PROGRAM MAIN
VAR
	rWriteAnalog1 : REAL;
	rWriteAnalog2 : REAL;
END_VAR

GVL.bAnalog_Outputs[1] := REAL_TO_INT((rWriteAnalog1-4)/16*32767);
GVL.bAnalog_Outputs[2] := REAL_TO_INT((rWriteAnalog2-4)/16*32767);

END_PROGRAM

(* stored: Version 1.1.0.1, ProductVersion 3.1.4024.12
   POU MAIN: Id {e589d767-5060-4f5a-94e2-37fc12fad615}, SpecialFunc None *)
